// TIA Portal V17 export
// export: Created 2021-12-03T08:12:53.3724713Z, ExportSetting WithDefaults, DisplayName Totally Integrated Automation Portal, DisplayVersion V17, DisplayName TIA Portal Openness, DisplayVersion V17, DisplayName TIA Portal Version Control Interface, DisplayVersion V17, DisplayName STEP 7 Professional, DisplayVersion V17, DisplayName STEP 7 Safety, DisplayVersion V17, DisplayName WinCC Advanced, DisplayVersion V17
DATA_BLOCK "GDB_HmiTestBtns"   // DB1003
VERSION : 0.1
// stored: AutoNumber false, IsOnlyStoredInLoadMemory false, IsWriteProtectedInAS false
   VAR
      TB1_00_Mod400V : Bool;   // 1Q3 Контактор модулятор 400В
      TB1_01_Chill : Bool;   // 1Q5 Чиллер
      TB1_02_Conveyor : Bool;   // 1Q7 Частортный преобразователь
      TB1_03_AccCons : Bool;   // 2Q3 Консоль ускорителя
      TB1_04_Acc : Bool;   // 2Q7 Ускоритель
      TB1_05_Mod230V : Bool;   // 3Q3 Модулятор 230В
      TB1_06_IntrlcAcc : Bool;   // 4A1 Интерлок ускорителя
      TB1_07_TstLmp : Bool;   // Тест ламп
      TB1_08_ConvFwrd : Bool;   // Перемещение вперед
      TB1_09_ConvBwrd : Bool;   // Перемещение назад
      TB1_10_DetLineStrt : Bool;   // Старт дет. линейки
      TB1_11_DetLineStp : Bool;   // Стоп дет. линейки
      TB1_12_DetLineSetup : Bool;   // Установка параметров дет. линейки
      TB1_13_StnDfltRst : Bool;   // Сброс настроек по умолчанию
      TB1_14_ChilVlv : Bool;   // Клапан чиллера
      TB1_15_ModSwit : Bool;   // Переключатель модулятора
      TB2_00_AccRst : Bool;   // Сброс на ускоритель
      TB2_01_AccWarm : Bool;   // Запрос прогрева для ускорителя
      TB2_02_AccWarnFull : Bool;   // Запрос на выход из паузы ускорителя
      TB2_03_AccXRay : Bool;   // Запрос на включение излучения
      TB2_04_AccChgDose : Bool;   // Запрос на смену дозы
      TB2_05_AccRfOn : Bool;   // Включение СВЧ
      TB2_06_HornTst : Bool;   // Тест сирены
      TB2_07_ConvSpdCount : Bool;   // Подсчет скорости конвйера
      TB2_08_StrtSpdCount : Bool;   // Запуск подсчета фактической скорости
      TB2_09_ : Bool;
      TB2_10_ : Bool;
      TB2_11_ : Bool;
      TB2_12_ : Bool;
      TB2_13_ : Bool;
      TB2_14_ : Bool;
      TB2_15_ : Bool;
   END_VAR
BEGIN
END_DATA_BLOCK
